TYPE ST_Z4_Params :
STRUCT
	tDrilling	:	TIME	:= T#4S;	// durata della fase di foratura
	tDelayToZ5	:	TIME	:= T#1S;	// ritardo per arrivare a Z5
	tStopDelay	:	TIME	:= T#1S;	// permanenza nello stato Stop
	tRecovering :   TIME	:= T#2S;
END_STRUCT
END_TYPE

(* stored: Version 1.1.0.1
   DUT ST_Z4_Params: Id {79853cb3-3690-0ee8-20a0-8a75ebc3147d} *)
